INTERFACE I_OwnedComp EXTENDS I_Component

PROPERTY Owner : I_CompRegister
GET
END_GET
END_PROPERTY

END_INTERFACE

(* stored: Version 1.1.0.1
   Itf I_OwnedComp: Id {76d104c7-8c2d-456d-8e4c-3ee26ed6ed8c}
   Property Owner: Id {5ef96ad3-5959-4641-a1c9-55a440b9aad2}
   Get Get: Id {83d3b527-0a7f-46eb-affa-ce3115ce7a7e} *)
